(* Logix 5000 project; controller CarbonScout_MK6 vendor 1 type 14 code 154 rev 32.11; software revision 32.00; part 9 of 17 *)
(* tags used below, declared in another part *)
   AI_AIT_01 : P_AIn;   // pH
   AI_AIT_02 : P_AIn;   // DO
   AI_FIT_01 : P_AIn;   // Purge water flow
   AI_LIT_01 : P_AIn;   // Carbon Scout Laser Level Transmitter
   AI_LIT_02 : P_AIn;   // Carbon Scout Cone Level Transmitter
   AI_PIT_01 : P_AIn;   // Water supply pressure
   AI_WIT_01 : P_AIn;   // Weight measure
   CS_Alarms : P_Alarm[80];
   CS_DINTParams : DINT[100];
   CS_EventNum : DINT;
   CS_Result : CS_Results;   // Sample Result Live Async
   CS_Rules : DINT[17];
   CS_SampleSeq : DINT[129];
   CS_Seq : GEK_Sequence;
   CS_SeqCheckSum1 : DINT;
   CS_SeqCheckSum2 : DINT;
   CS_Tank : CS_TankParams[20];
   CS_TankOrder : DINT[17];
   CS_Timer : TIMER[80];
   CS_XRF : XRF;
   N50 : DINT[20];   // Out To Client (Ready only)
   N51 : DINT[5];   // From Client
   Oneshot : DINT;
   TankPointer : DINT;
   TimeAndDate : DINT[7];
   Valve_SPR_01 : P_ValveSO;   // Air injection valve
   Valve_XV_01 : P_ValveSO;   // Sample Valve Tank 1
   Valve_XV_02 : P_ValveSO;   // Sample Valve Tank 2
   Valve_XV_03 : P_ValveSO;   // Sample Valve Tank 3
   Valve_XV_04 : P_ValveSO;   // Sample Valve Tank 4
   Valve_XV_05 : P_ValveSO;   // Sample Valve Tank 5
   Valve_XV_06 : P_ValveSO;   // Sample Valve Tank 6
   Valve_XV_07 : P_ValveSO;   // Sample Valve Tank 7
   Valve_XV_08 : P_ValveSO;   // Sample Valve Tank 8
   Valve_XV_09 : P_ValveSO;   // Sample Valve Tank 9
   Valve_XV_10 : P_ValveSO;   // Sample Valve Tank 10
   Valve_XV_11 : P_ValveSO;   // Purge Valve
   Valve_XV_12 : P_ValveSO;   // Slurry inlet vavle
   Valve_XV_13 : P_ValveSO;   // Sample line vavle
   Valve_XV_14 : P_ValveSO;   // Top wash vavle
   Valve_XV_15 : P_ValveSO;   // Bottme wash vavle
   Valve_XV_16 : P_ValveSO;   // Potable water valve / Supply Water Valve
   Valve_XV_17 : P_ValveSO;   // Sample cone outlet vavle
   Valve_XV_18 : P_ValveSO;   // Sample strainer discharge
   Valve_XV_19 : P_ValveSO;   // Laser window
   Valve_XV_21_30 : P_ValveSO;   // Sample isolation valve
   Valve_XV_30 : P_ValveSO;   // XRF cooling valve
   Valve_XV_40 : P_ValveSO;   // XRF power on valve
(* DataMapping, continued *)

ROUTINE InputMapping   (* ladder *)
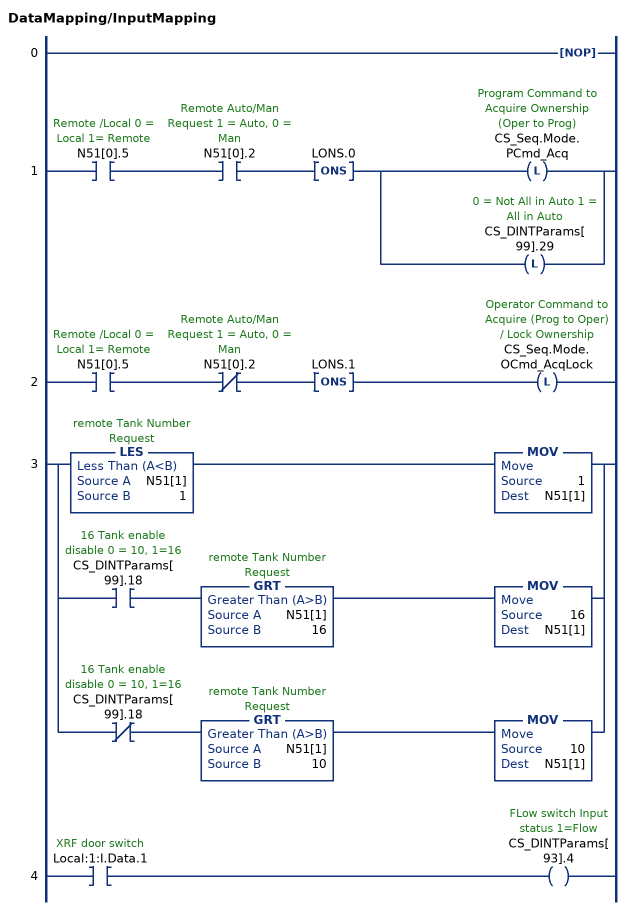
   0: NOP();
   1: XIC(N51[0].5)XIC(N51[0].2)ONS(LONS.0)[OTL(CS_Seq.Mode.PCmd_Acq) ,OTL(CS_DINTParams[99].29) ];
   2: XIC(N51[0].5)XIO(N51[0].2)ONS(LONS.1)OTL(CS_Seq.Mode.OCmd_AcqLock);
   3: [LES(N51[1],1) MOV(1,N51[1]) ,XIC(CS_DINTParams[99].18) GRT(N51[1],16) MOV(16,N51[1]) ,XIO(CS_DINTParams[99].18) GRT(N51[1],10) MOV(10,N51[1]) ];
   4: XIC(Local:1:I.Data.1)OTE(CS_DINTParams[93].4);
END_ROUTINE

ROUTINE Main   (* ladder *)
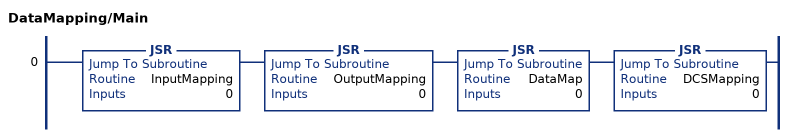
   0: JSR(InputMapping,0)JSR(OutputMapping,0)JSR(DataMap,0)JSR(DCSMapping,0);
END_ROUTINE

ROUTINE OutputMapping   (* ladder *)
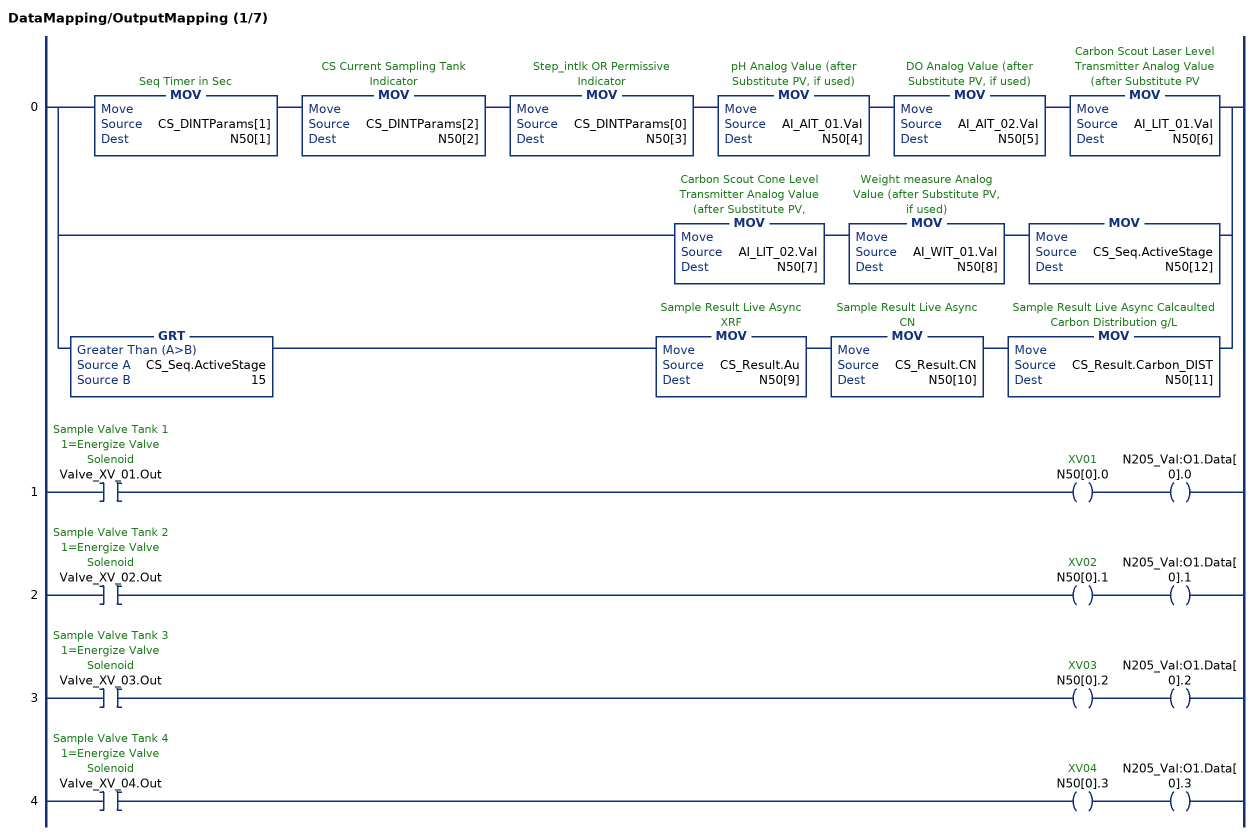
   0: [MOV(CS_DINTParams[1],N50[1]) MOV(CS_DINTParams[2],N50[2]) MOV(CS_DINTParams[0],N50[3]) MOV(AI_AIT_01.Val,N50[4]) MOV(AI_AIT_02.Val,N50[5]) MOV(AI_LIT_01.Val,N50[6]) ,MOV(AI_LIT_02.Val,N50[7]) MOV(AI_WIT_01.Val,N50[8]) MOV(CS_Seq.ActiveStage,N50[12]) ,GRT(CS_Seq.ActiveStage,15) MOV(CS_Result.Au,N50[9]) MOV(CS_Result.CN,N50[10]) MOV(CS_Result.Carbon_DIST,N50[11]) ];
   1: XIC(Valve_XV_01.Out)OTE(N50[0].0)OTE(N205_Val:O1.Data[0].0);
   2: XIC(Valve_XV_02.Out)OTE(N50[0].1)OTE(N205_Val:O1.Data[0].1);
   3: XIC(Valve_XV_03.Out)OTE(N50[0].2)OTE(N205_Val:O1.Data[0].2);
   4: XIC(Valve_XV_04.Out)OTE(N50[0].3)OTE(N205_Val:O1.Data[0].3);
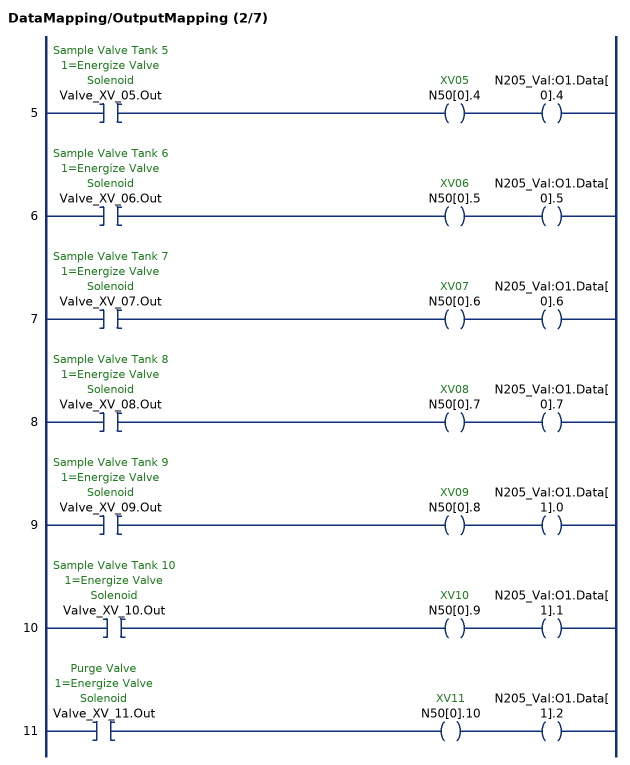
   5: XIC(Valve_XV_05.Out)OTE(N50[0].4)OTE(N205_Val:O1.Data[0].4);
   6: XIC(Valve_XV_06.Out)OTE(N50[0].5)OTE(N205_Val:O1.Data[0].5);
   7: XIC(Valve_XV_07.Out)OTE(N50[0].6)OTE(N205_Val:O1.Data[0].6);
   8: XIC(Valve_XV_08.Out)OTE(N50[0].7)OTE(N205_Val:O1.Data[0].7);
   9: XIC(Valve_XV_09.Out)OTE(N50[0].8)OTE(N205_Val:O1.Data[1].0);
   10: XIC(Valve_XV_10.Out)OTE(N50[0].9)OTE(N205_Val:O1.Data[1].1);
   11: XIC(Valve_XV_11.Out)OTE(N50[0].10)OTE(N205_Val:O1.Data[1].2);
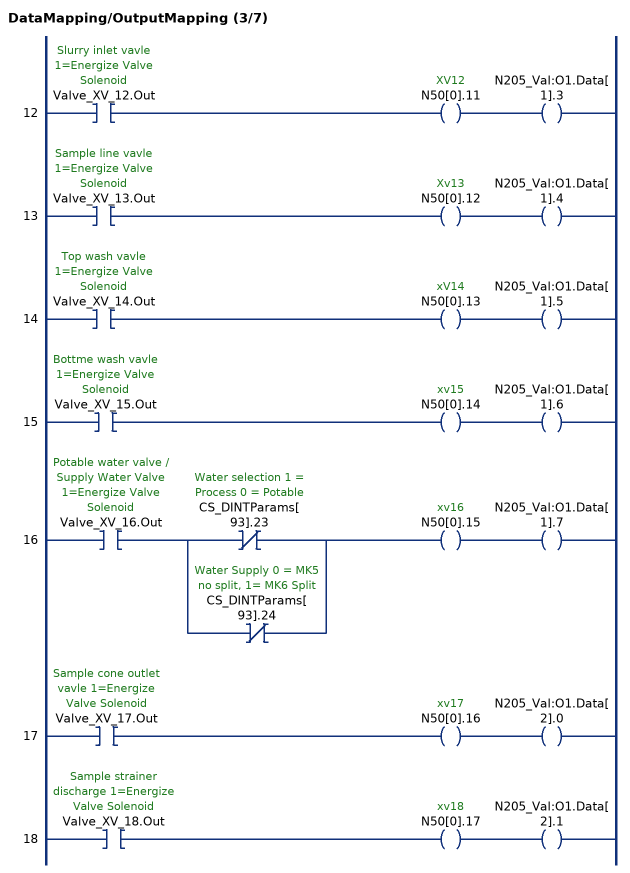
   12: XIC(Valve_XV_12.Out)OTE(N50[0].11)OTE(N205_Val:O1.Data[1].3);
   13: XIC(Valve_XV_13.Out)OTE(N50[0].12)OTE(N205_Val:O1.Data[1].4);
   14: XIC(Valve_XV_14.Out)OTE(N50[0].13)OTE(N205_Val:O1.Data[1].5);
   15: XIC(Valve_XV_15.Out)OTE(N50[0].14)OTE(N205_Val:O1.Data[1].6);
   16: XIC(Valve_XV_16.Out)[XIO(CS_DINTParams[93].23) ,XIO(CS_DINTParams[93].24) ]OTE(N50[0].15)OTE(N205_Val:O1.Data[1].7);
   17: XIC(Valve_XV_17.Out)OTE(N50[0].16)OTE(N205_Val:O1.Data[2].0);
   18: XIC(Valve_XV_18.Out)OTE(N50[0].17)OTE(N205_Val:O1.Data[2].1);
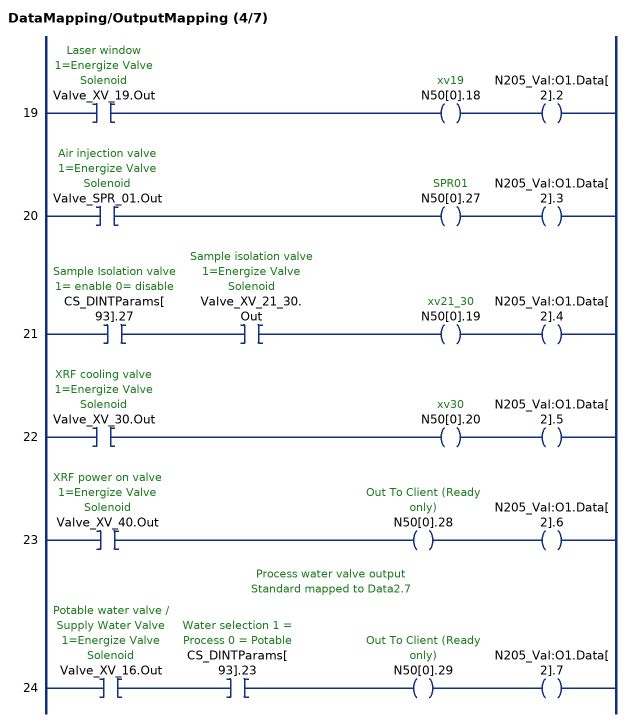
   19: XIC(Valve_XV_19.Out)OTE(N50[0].18)OTE(N205_Val:O1.Data[2].2);
   20: XIC(Valve_SPR_01.Out)OTE(N50[0].27)OTE(N205_Val:O1.Data[2].3);
   21: XIC(CS_DINTParams[93].27)XIC(Valve_XV_21_30.Out)OTE(N50[0].19)OTE(N205_Val:O1.Data[2].4);
   22: XIC(Valve_XV_30.Out)OTE(N50[0].20)OTE(N205_Val:O1.Data[2].5);
   23: XIC(Valve_XV_40.Out)OTE(N50[0].28)OTE(N205_Val:O1.Data[2].6);
   // Process water valve output
   // Standard mapped to Data2.7
   24: XIC(Valve_XV_16.Out)XIC(CS_DINTParams[93].23)OTE(N50[0].29)OTE(N205_Val:O1.Data[2].7);
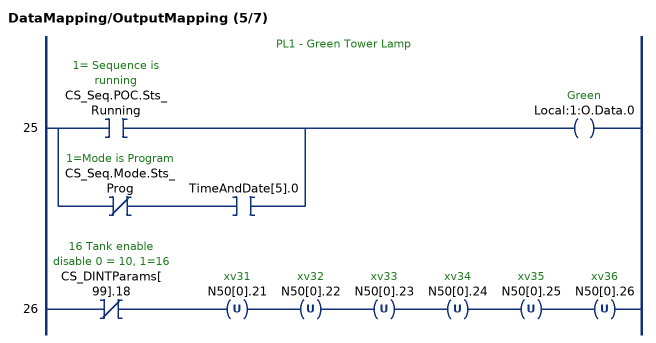
   // PL1 - Green Tower Lamp
   25: [XIC(CS_Seq.POC.Sts_Running) ,XIO(CS_Seq.Mode.Sts_Prog) XIC(TimeAndDate[5].0) ]OTE(Local:1:O.Data.0);
   26: XIO(CS_DINTParams[99].18)OTU(N50[0].21)OTU(N50[0].22)OTU(N50[0].23)OTU(N50[0].24)OTU(N50[0].25)OTU(N50[0].26);
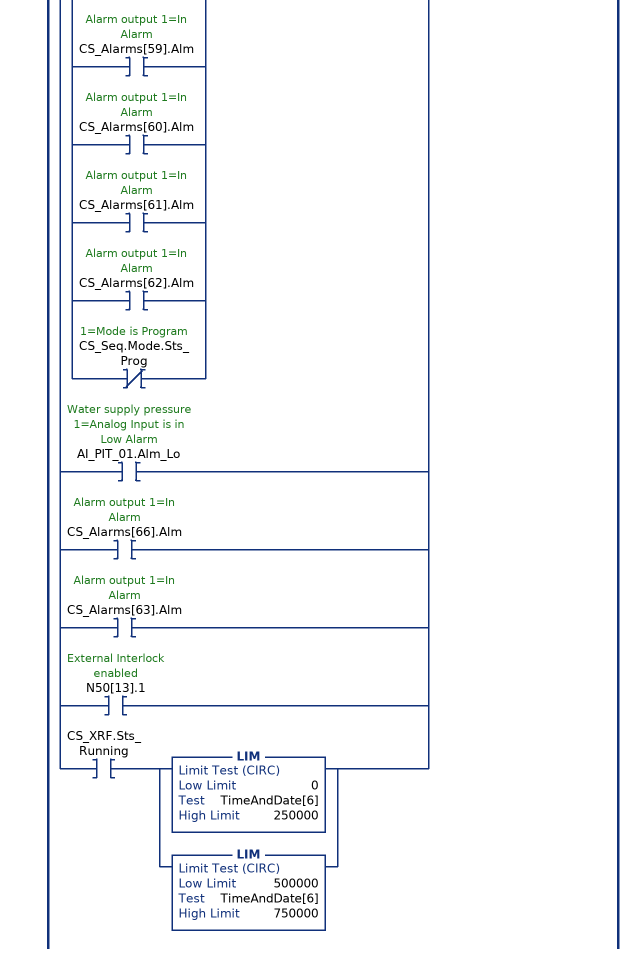
   // PL2 - Amber Tower Lamp
   27: [[XIC(CS_Alarms[24].Alm) ,XIC(CS_Alarms[14].Inp) ,XIC(CS_Alarms[15].Alm) ,XIC(CS_Alarms[16].Alm) ,XIC(CS_Alarms[17].Alm) ,XIC(CS_Alarms[18].Alm) ,XIC(CS_Alarms[19].Alm) ,XIC(CS_Alarms[20].Alm) ,XIC(CS_Alarms[21].Alm) ,XIC(CS_Alarms[22].Alm) ,XIC(CS_Alarms[23].Alm) ,XIC(CS_Alarms[57].Alm) ,XIC(CS_Alarms[58].Alm) ,XIC(CS_Alarms[59].Alm) ,XIC(CS_Alarms[60].Alm) ,XIC(CS_Alarms[61].Alm) ,XIC(CS_Alarms[62].Alm) ,XIO(CS_Seq.Mode.Sts_Prog) ] XIC(TimeAndDate[5].0) XIO(CS_XRF.Sts_Running) ,XIC(AI_PIT_01.Alm_Lo) ,XIC(CS_Alarms[66].Alm) ,XIC(CS_Alarms[63].Alm) ,XIC(N50[13].1) ,XIC(CS_XRF.Sts_Running) [LIM(0,TimeAndDate[6],250000) ,LIM(500000,TimeAndDate[6],750000) ] ]OTE(Local:1:O.Data.1);
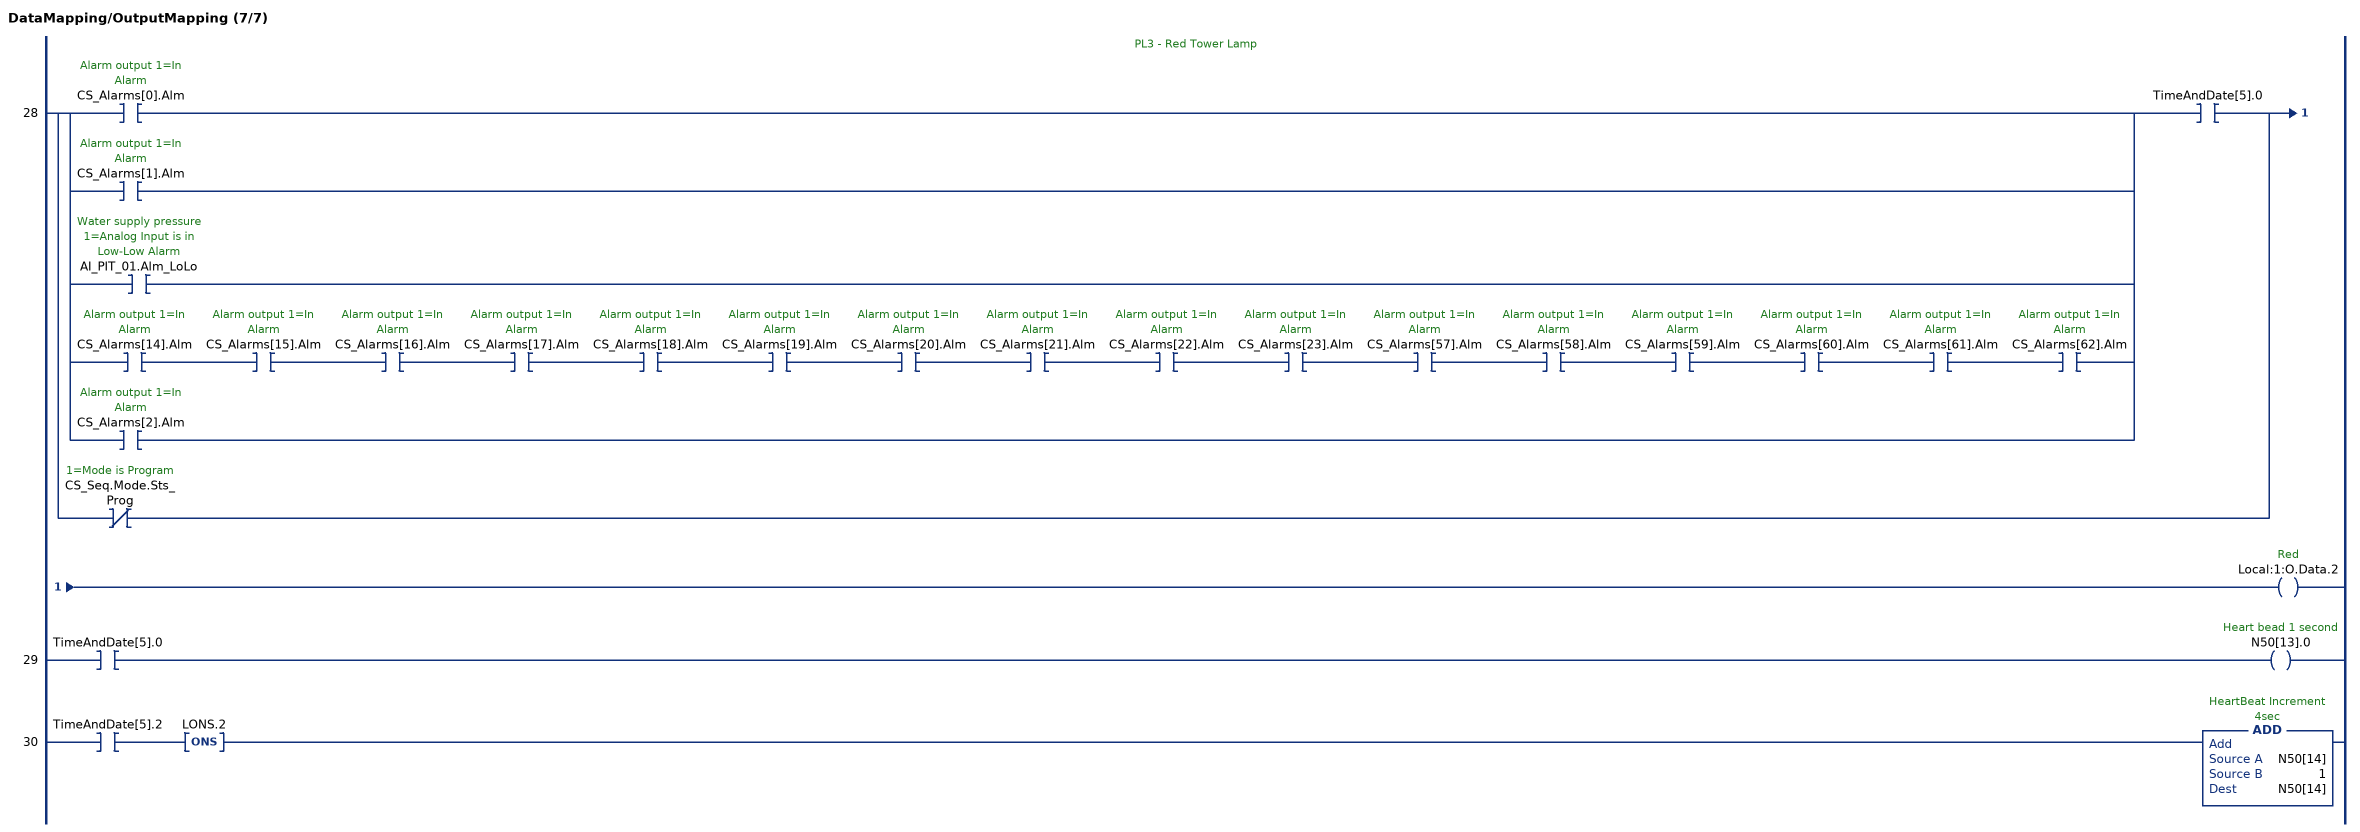
   // PL3 - Red Tower Lamp
   28: [[XIC(CS_Alarms[0].Alm) ,XIC(CS_Alarms[1].Alm) ,XIC(AI_PIT_01.Alm_LoLo) ,XIC(CS_Alarms[14].Alm) XIC(CS_Alarms[15].Alm) XIC(CS_Alarms[16].Alm) XIC(CS_Alarms[17].Alm) XIC(CS_Alarms[18].Alm) XIC(CS_Alarms[19].Alm) XIC(CS_Alarms[20].Alm) XIC(CS_Alarms[21].Alm) XIC(CS_Alarms[22].Alm) XIC(CS_Alarms[23].Alm) XIC(CS_Alarms[57].Alm) XIC(CS_Alarms[58].Alm) XIC(CS_Alarms[59].Alm) XIC(CS_Alarms[60].Alm) XIC(CS_Alarms[61].Alm) XIC(CS_Alarms[62].Alm) ,XIC(CS_Alarms[2].Alm) ] XIC(TimeAndDate[5].0) ,XIO(CS_Seq.Mode.Sts_Prog) ]OTE(Local:1:O.Data.2);
   29: XIC(TimeAndDate[5].0)OTE(N50[13].0);
   30: XIC(TimeAndDate[5].2)ONS(LONS.2)ADD(N50[14],1,N50[14]);
END_ROUTINE
END_PROGRAM

PROGRAM Powerup   (* main routine Yes *)
VAR
   ControllerFaultReset : DINT;
   MajorFaultBit : DINT;
   MajorFaultEvent : DINT;
   MinorEvents : DINT;
   MinorFaultBits : DINT;
END_VAR

ROUTINE Yes   (* ladder *)
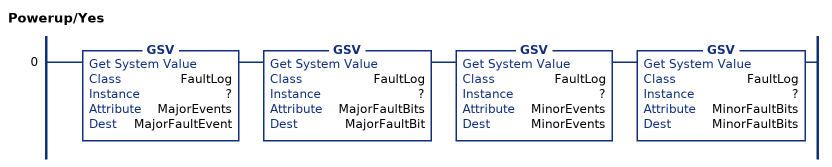
   0: GSV(FaultLog,?,MajorEvents,MajorFaultEvent)GSV(FaultLog,?,MajorFaultBits,MajorFaultBit)GSV(FaultLog,?,MinorEvents,MinorEvents)GSV(FaultLog,?,MinorFaultBits,MinorFaultBits);
END_ROUTINE
END_PROGRAM

PROGRAM SeqProgram   (* main routine MainRoutine *)
VAR
   CNT : DINT := 311;
   CS_EVentNumStore : DINT := 1;
   Data_TLSaver : BOOL := 1;
   Delay : TIMER := (PRE := 10000);
   DN_Cal : BOOL;   // Calculation Done Bit to proceed next step
   EventDone : BOOL;
   ExtraValveCNTReached : BOOL; {access Read Only}
   ExtraValvesAuto : BOOL; {access Read Only}
   i : DINT;
   Index : DINT := 1;
   IndexNumStore : DINT := 8;
   InitialPurgeRequired : BOOL := 1;
   LIT_Prev : REAL := 1441.9149;
   LocalSampleTank : DINT := 6;
   LOnlineNumber : DINT := 7;
   LONS : DINT := 1;
   ManualRunning : BOOL;
   MaxFindIndexNum : DINT := 16;
   MaxFindNum : DINT := 1;
   ONS : BOOL[32] := ([1] := 1, [4] := 1);
   SampleIndexNum : DINT := 8;
   SampleIndexNum2 : DINT;
   SONS : DINT := 511;
   storage : BOOL;
   TankDiagnosticCheck : BOOL;
   TimeCompare : TimerCompare := (In_PresetTime1_Multiplier := 60, In_PresetTime2 := 10, In_PresetTime2_Multiplier := 1, In_ActiveStep := 23);
   TimeRemainingCal : TimeRemainingCal := (In_PresetTime := 30, RemainingSec := 8, In_Time := 1);
   XRF_DirtyWinCounter : COUNTER := (PRE := 10);
   XRF_ReadyTimer : TIMER := (PRE := 10000);
END_VAR

ROUTINE _SampleSeq   (* ladder *)
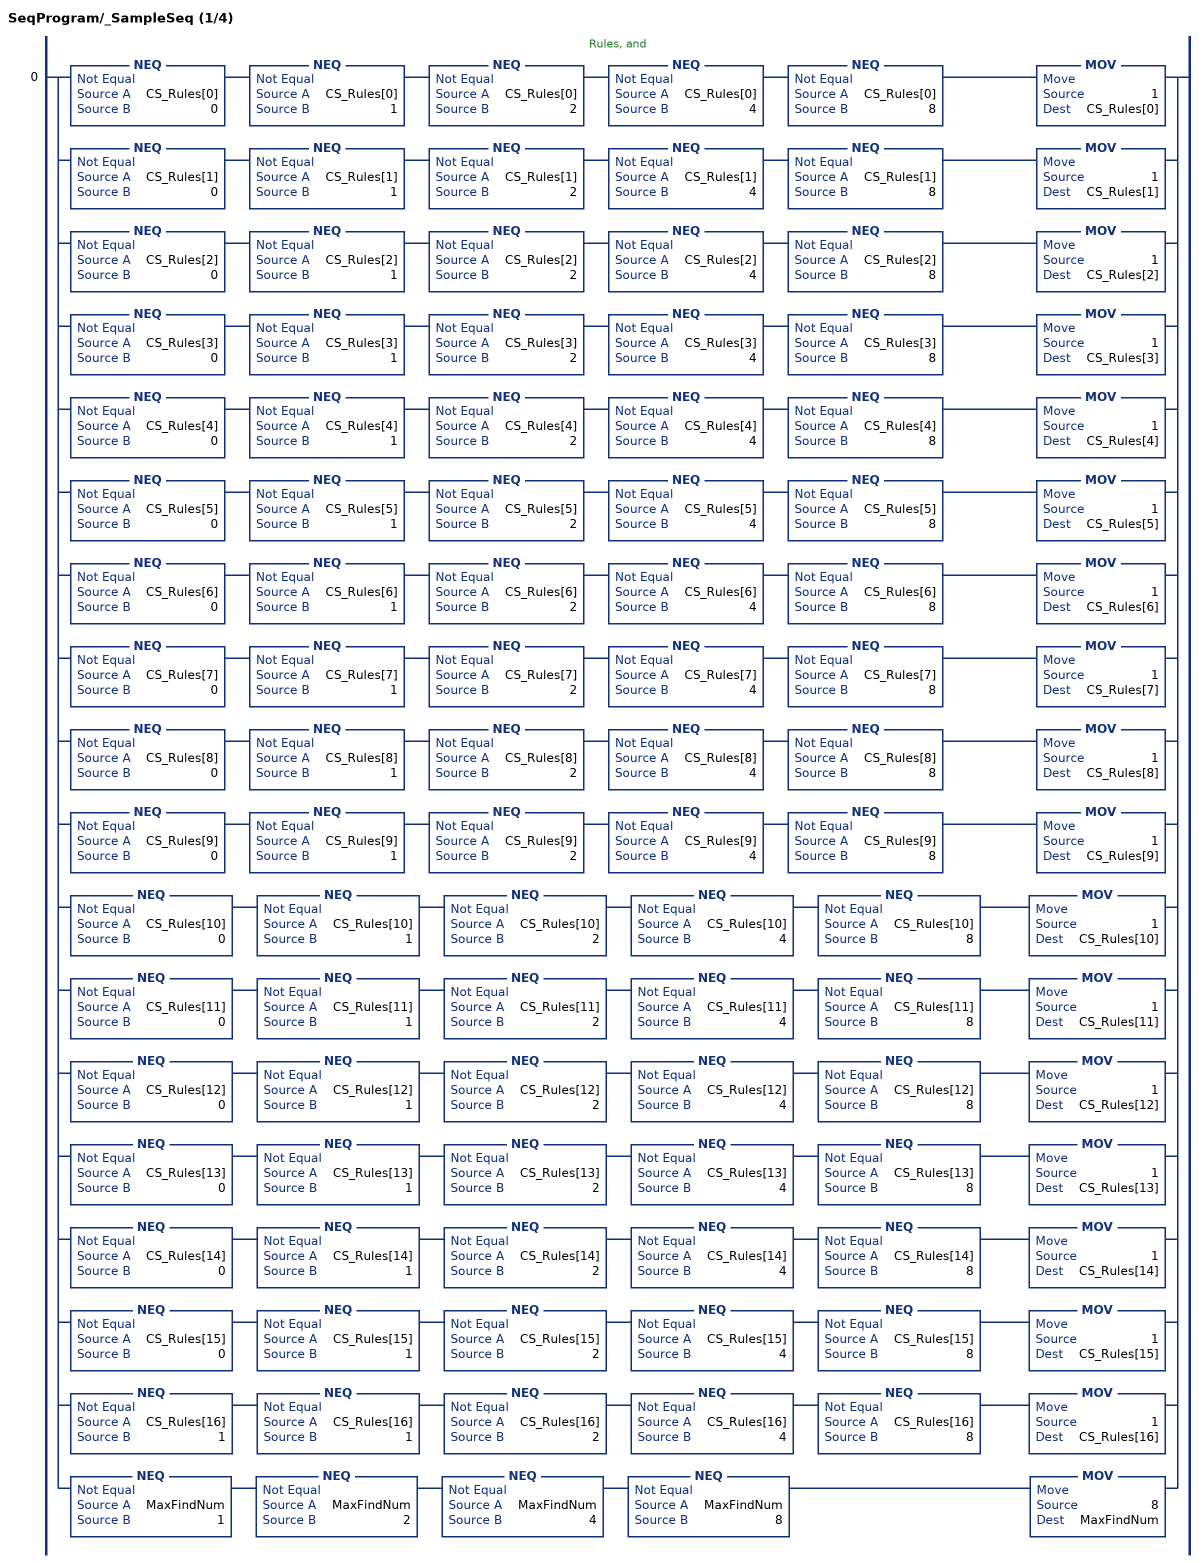
   // Rules, and
   0: [NEQ(CS_Rules[0],0) NEQ(CS_Rules[0],1) NEQ(CS_Rules[0],2) NEQ(CS_Rules[0],4) NEQ(CS_Rules[0],8) MOV(1,CS_Rules[0]) ,NEQ(CS_Rules[1],0) NEQ(CS_Rules[1],1) NEQ(CS_Rules[1],2) NEQ(CS_Rules[1],4) NEQ(CS_Rules[1],8) MOV(1,CS_Rules[1]) ,NEQ(CS_Rules[2],0) NEQ(CS_Rules[2],1) NEQ(CS_Rules[2],2) NEQ(CS_Rules[2],4) NEQ(CS_Rules[2],8) MOV(1,CS_Rules[2]) ,NEQ(CS_Rules[3],0) NEQ(CS_Rules[3],1) NEQ(CS_Rules[3],2) NEQ(CS_Rules[3],4) NEQ(CS_Rules[3],8) MOV(1,CS_Rules[3]) ,NEQ(CS_Rules[4],0) NEQ(CS_Rules[4],1) NEQ(CS_Rules[4],2) NEQ(CS_Rules[4],4) NEQ(CS_Rules[4],8) MOV(1,CS_Rules[4]) ,NEQ(CS_Rules[5],0) NEQ(CS_Rules[5],1) NEQ(CS_Rules[5],2) NEQ(CS_Rules[5],4) NEQ(CS_Rules[5],8) MOV(1,CS_Rules[5]) ,NEQ(CS_Rules[6],0) NEQ(CS_Rules[6],1) NEQ(CS_Rules[6],2) NEQ(CS_Rules[6],4) NEQ(CS_Rules[6],8) MOV(1,CS_Rules[6]) ,NEQ(CS_Rules[7],0) NEQ(CS_Rules[7],1) NEQ(CS_Rules[7],2) NEQ(CS_Rules[7],4) NEQ(CS_Rules[7],8) MOV(1,CS_Rules[7]) ,NEQ(CS_Rules[8],0) NEQ(CS_Rules[8],1) NEQ(CS_Rules[8],2) NEQ(CS_Rules[8],4) NEQ(CS_Rules[8],8) MOV(1,CS_Rules[8]) ,NEQ(CS_Rules[9],0) NEQ(CS_Rules[9],1) NEQ(CS_Rules[9],2) NEQ(CS_Rules[9],4) NEQ(CS_Rules[9],8) MOV(1,CS_Rules[9]) ,NEQ(CS_Rules[10],0) NEQ(CS_Rules[10],1) NEQ(CS_Rules[10],2) NEQ(CS_Rules[10],4) NEQ(CS_Rules[10],8) MOV(1,CS_Rules[10]) ,NEQ(CS_Rules[11],0) NEQ(CS_Rules[11],1) NEQ(CS_Rules[11],2) NEQ(CS_Rules[11],4) NEQ(CS_Rules[11],8) MOV(1,CS_Rules[11]) ,NEQ(CS_Rules[12],0) NEQ(CS_Rules[12],1) NEQ(CS_Rules[12],2) NEQ(CS_Rules[12],4) NEQ(CS_Rules[12],8) MOV(1,CS_Rules[12]) ,NEQ(CS_Rules[13],0) NEQ(CS_Rules[13],1) NEQ(CS_Rules[13],2) NEQ(CS_Rules[13],4) NEQ(CS_Rules[13],8) MOV(1,CS_Rules[13]) ,NEQ(CS_Rules[14],0) NEQ(CS_Rules[14],1) NEQ(CS_Rules[14],2) NEQ(CS_Rules[14],4) NEQ(CS_Rules[14],8) MOV(1,CS_Rules[14]) ,NEQ(CS_Rules[15],0) NEQ(CS_Rules[15],1) NEQ(CS_Rules[15],2) NEQ(CS_Rules[15],4) NEQ(CS_Rules[15],8) MOV(1,CS_Rules[15]) ,NEQ(CS_Rules[16],1) NEQ(CS_Rules[16],1) NEQ(CS_Rules[16],2) NEQ(CS_Rules[16],4) NEQ(CS_Rules[16],8) MOV(1,CS_Rules[16]) ,NEQ(MaxFindNum,1) NEQ(MaxFindNum,2) NEQ(MaxFindNum,4) NEQ(MaxFindNum,8) MOV(8,MaxFindNum) ];
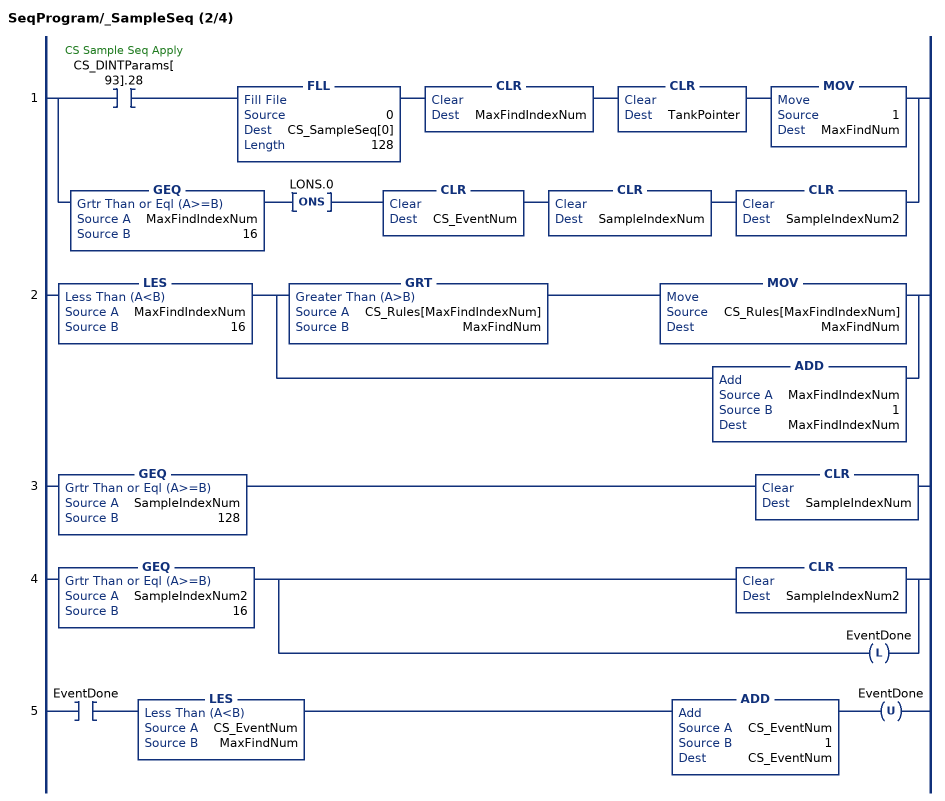
   1: [XIC(CS_DINTParams[93].28) FLL(0,CS_SampleSeq[0],128) CLR(MaxFindIndexNum) CLR(TankPointer) MOV(1,MaxFindNum) ,GEQ(MaxFindIndexNum,16) ONS(LONS.0) CLR(CS_EventNum) CLR(SampleIndexNum) CLR(SampleIndexNum2) ];
   2: LES(MaxFindIndexNum,16)[GRT(CS_Rules[MaxFindIndexNum],MaxFindNum) MOV(CS_Rules[MaxFindIndexNum],MaxFindNum) ,ADD(MaxFindIndexNum,1,MaxFindIndexNum) ];
   3: GEQ(SampleIndexNum,128)CLR(SampleIndexNum);
   4: GEQ(SampleIndexNum2,16)[CLR(SampleIndexNum2) ,OTL(EventDone) ];
   5: XIC(EventDone)LES(CS_EventNum,MaxFindNum)ADD(CS_EventNum,1,CS_EventNum)OTU(EventDone);
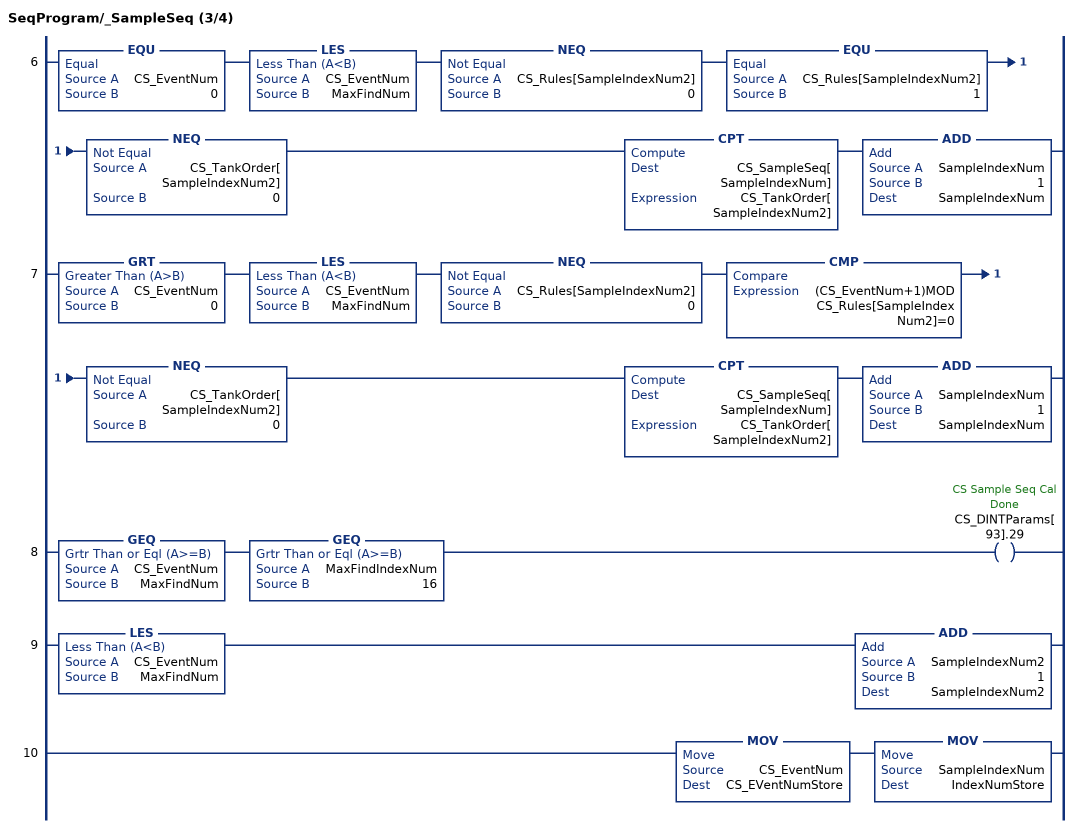
   6: EQU(CS_EventNum,0)LES(CS_EventNum,MaxFindNum)NEQ(CS_Rules[SampleIndexNum2],0)EQU(CS_Rules[SampleIndexNum2],1)NEQ(CS_TankOrder[SampleIndexNum2],0)CPT(CS_SampleSeq[SampleIndexNum],CS_TankOrder[SampleIndexNum2])ADD(SampleIndexNum,1,SampleIndexNum);
   7: GRT(CS_EventNum,0)LES(CS_EventNum,MaxFindNum)NEQ(CS_Rules[SampleIndexNum2],0)CMP((CS_EventNum+1)MOD CS_Rules[SampleIndexNum2]=0)NEQ(CS_TankOrder[SampleIndexNum2],0)CPT(CS_SampleSeq[SampleIndexNum],CS_TankOrder[SampleIndexNum2])ADD(SampleIndexNum,1,SampleIndexNum);
   8: GEQ(CS_EventNum,MaxFindNum)GEQ(MaxFindIndexNum,16)OTE(CS_DINTParams[93].29);
   9: LES(CS_EventNum,MaxFindNum)ADD(SampleIndexNum2,1,SampleIndexNum2);
   10: MOV(CS_EventNum,CS_EVentNumStore)MOV(SampleIndexNum,IndexNumStore);
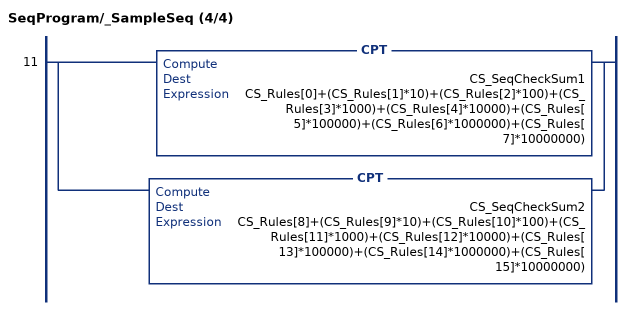
   11: [CPT(CS_SeqCheckSum1,CS_Rules[0]+(CS_Rules[1]*10)+(CS_Rules[2]*100)+(CS_Rules[3]*1000)+(CS_Rules[4]*10000)+(CS_Rules[5]*100000)+(CS_Rules[6]*1000000)+(CS_Rules[7]*10000000)) ,CPT(CS_SeqCheckSum2,CS_Rules[8]+(CS_Rules[9]*10)+(CS_Rules[10]*100)+(CS_Rules[11]*1000)+(CS_Rules[12]*10000)+(CS_Rules[13]*100000)+(CS_Rules[14]*1000000)+(CS_Rules[15]*10000000)) ];
END_ROUTINE

ROUTINE Alarms   (* ladder *)
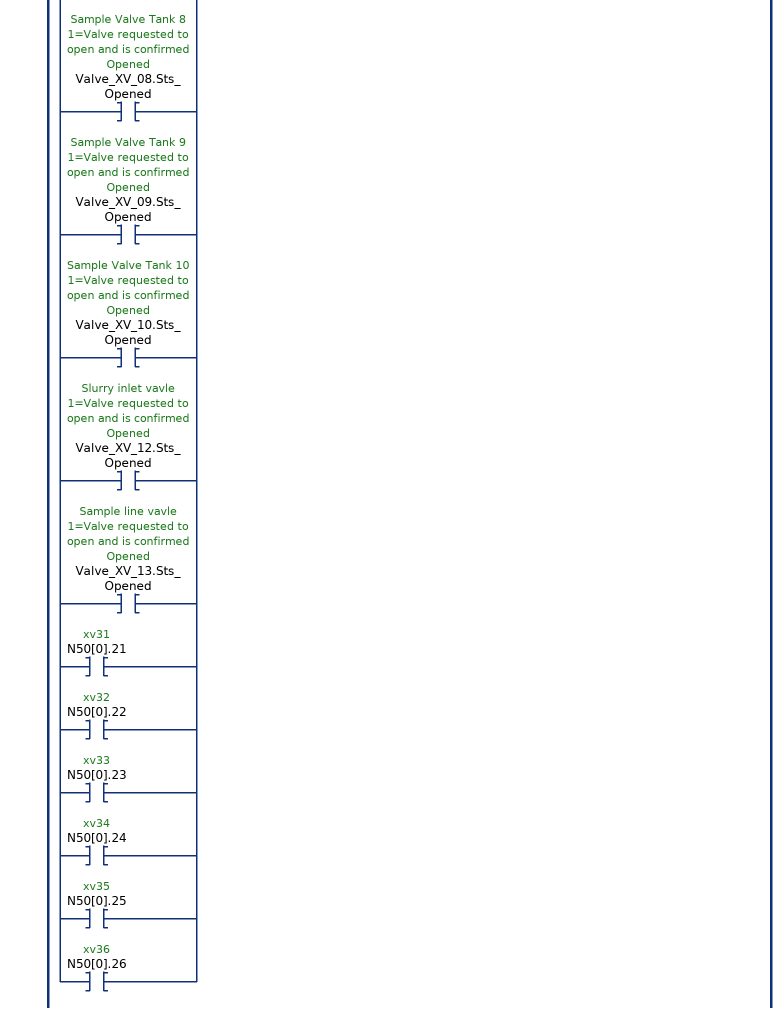
   0: [XIC(Valve_XV_01.Sts_Opened) ,XIC(Valve_XV_12.Sts_Opened) ,XIC(Valve_XV_02.Sts_Opened) ,XIC(Valve_XV_03.Sts_Opened) ,XIC(Valve_XV_04.Sts_Opened) ,XIC(Valve_XV_05.Sts_Opened) ,XIC(Valve_XV_06.Sts_Opened) ,XIC(Valve_XV_07.Sts_Opened) ,XIC(Valve_XV_08.Sts_Opened) ,XIC(Valve_XV_09.Sts_Opened) ,XIC(Valve_XV_10.Sts_Opened) ,XIC(Valve_XV_12.Sts_Opened) ,XIC(Valve_XV_13.Sts_Opened) ,XIC(N50[0].21) ,XIC(N50[0].22) ,XIC(N50[0].23) ,XIC(N50[0].24) ,XIC(N50[0].25) ,XIC(N50[0].26) ]XIC(Valve_XV_11.Sts_Opened)XIO(CS_DINTParams[93].0)OTE(AI_FIT_01.Inp_LoGate)OTE(AI_FIT_01.Inp_LoLoGate);
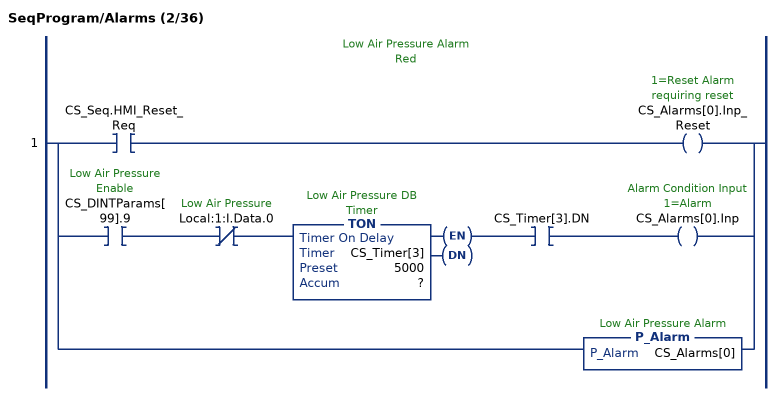
   // Low Air Pressure Alarm
   // Red
   1: [XIC(CS_Seq.HMI_Reset_Req) OTE(CS_Alarms[0].Inp_Reset) ,XIC(CS_DINTParams[99].9) XIO(Local:1:I.Data.0) TON(CS_Timer[3],?,?) XIC(CS_Timer[3].DN) OTE(CS_Alarms[0].Inp) ,P_Alarm(CS_Alarms[0]) ];
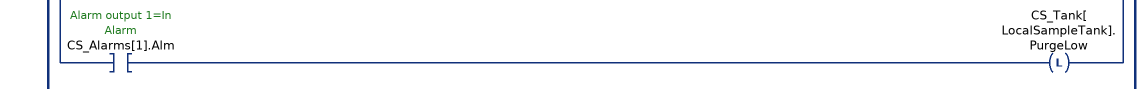
   // Purge Water Flow Alarm
   // Amber
   2: [XIC(CS_Seq.HMI_Reset_Req) OTE(CS_Alarms[1].Inp_Reset) ,[XIC(Valve_XV_01.Sts_Opened) ,XIC(Valve_XV_02.Sts_Opened) ,XIC(Valve_XV_03.Sts_Opened) ,XIC(Valve_XV_04.Sts_Opened) ,XIC(Valve_XV_05.Sts_Opened) ,XIC(Valve_XV_06.Sts_Opened) ,XIC(Valve_XV_07.Sts_Opened) ,XIC(Valve_XV_08.Sts_Opened) ,XIC(Valve_XV_09.Sts_Opened) ,XIC(Valve_XV_10.Sts_Opened) ,XIC(Valve_XV_12.Sts_Opened) ,XIC(Valve_XV_13.Sts_Opened) ,XIC(N50[0].21) ,XIC(N50[0].22) ,XIC(N50[0].23) ,XIC(N50[0].24) ,XIC(N50[0].25) ,XIC(N50[0].26) ] XIC(Valve_XV_11.Sts_Opened) [XIC(AI_FIT_01.Alm_Lo) XIO(CS_DINTParams[93].0) ,XIC(AI_FIT_01.Alm_LoLo) XIO(CS_DINTParams[93].0) ,XIO(Local:1:I.Data.1) XIC(CS_DINTParams[93].0) ] TON(CS_Timer[4],?,?) XIC(CS_Timer[4].DN) OTE(CS_Alarms[1].Inp) ,P_Alarm(CS_Alarms[1]) ,XIC(CS_Alarms[1].Alm) OTL(CS_Tank[LocalSampleTank].PurgeLow) ];
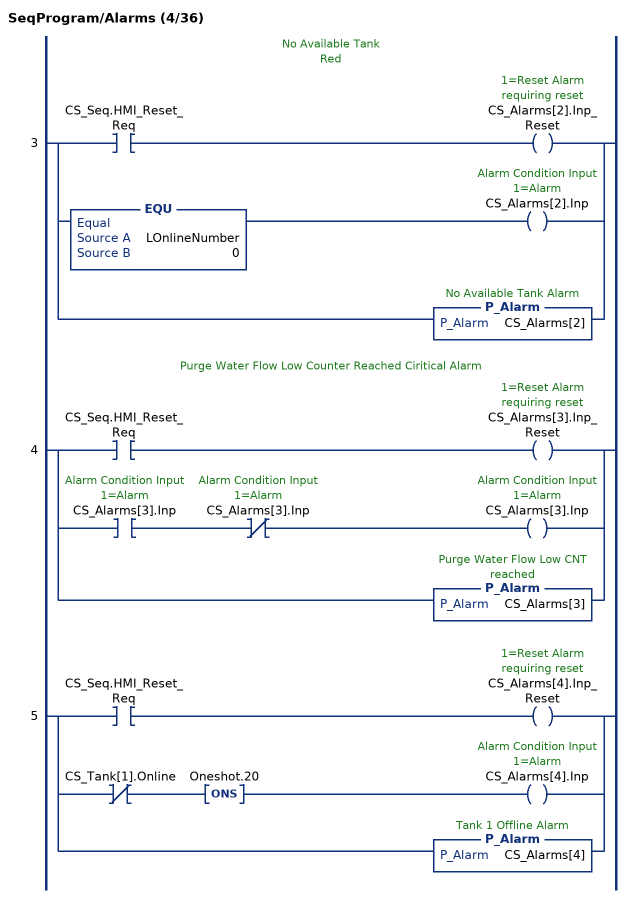
   // No Available Tank
   // Red
   3: [XIC(CS_Seq.HMI_Reset_Req) OTE(CS_Alarms[2].Inp_Reset) ,EQU(LOnlineNumber,0) OTE(CS_Alarms[2].Inp) ,P_Alarm(CS_Alarms[2]) ];
   // Purge Water Flow Low Counter Reached Ciritical Alarm
   4: [XIC(CS_Seq.HMI_Reset_Req) OTE(CS_Alarms[3].Inp_Reset) ,XIC(CS_Alarms[3].Inp) XIO(CS_Alarms[3].Inp) OTE(CS_Alarms[3].Inp) ,P_Alarm(CS_Alarms[3]) ];
   5: [XIC(CS_Seq.HMI_Reset_Req) OTE(CS_Alarms[4].Inp_Reset) ,XIO(CS_Tank[1].Online) ONS(Oneshot.20) OTE(CS_Alarms[4].Inp) ,P_Alarm(CS_Alarms[4]) ];
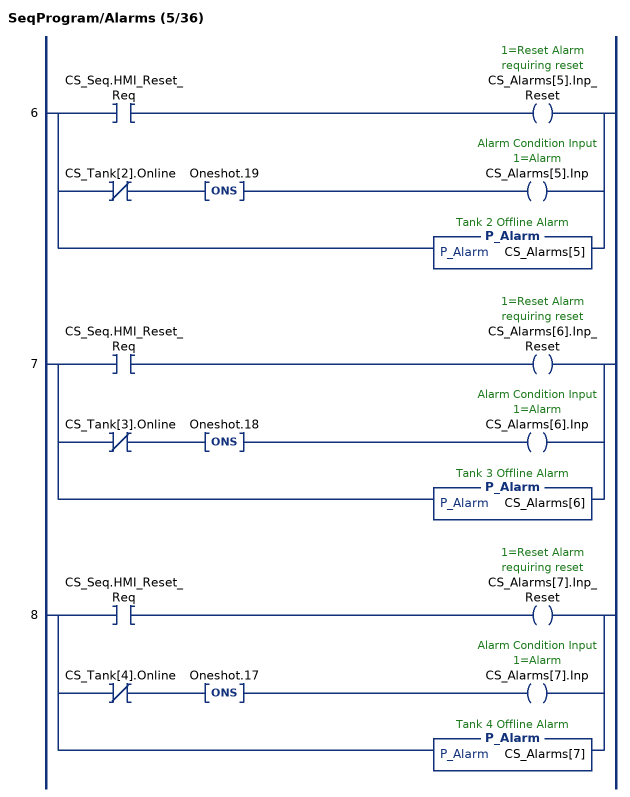
   6: [XIC(CS_Seq.HMI_Reset_Req) OTE(CS_Alarms[5].Inp_Reset) ,XIO(CS_Tank[2].Online) ONS(Oneshot.19) OTE(CS_Alarms[5].Inp) ,P_Alarm(CS_Alarms[5]) ];
   7: [XIC(CS_Seq.HMI_Reset_Req) OTE(CS_Alarms[6].Inp_Reset) ,XIO(CS_Tank[3].Online) ONS(Oneshot.18) OTE(CS_Alarms[6].Inp) ,P_Alarm(CS_Alarms[6]) ];
   8: [XIC(CS_Seq.HMI_Reset_Req) OTE(CS_Alarms[7].Inp_Reset) ,XIO(CS_Tank[4].Online) ONS(Oneshot.17) OTE(CS_Alarms[7].Inp) ,P_Alarm(CS_Alarms[7]) ];
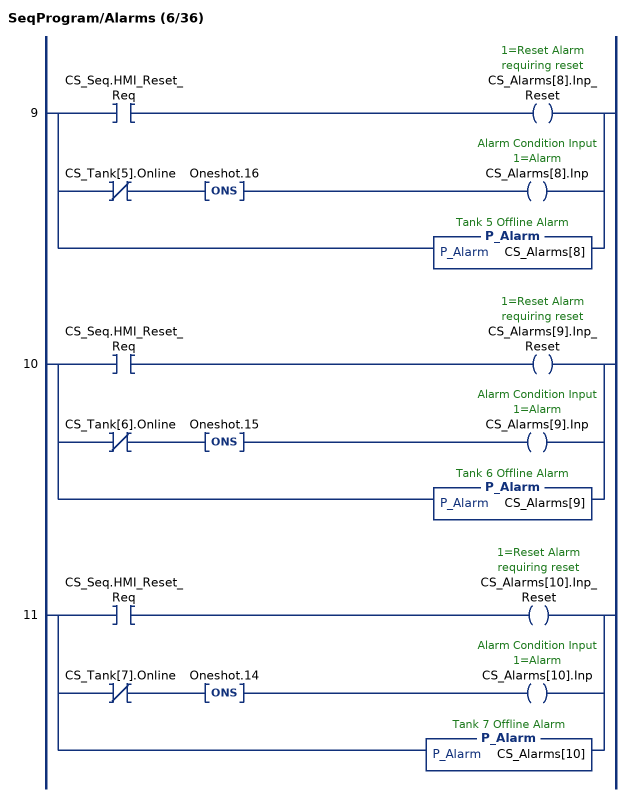
   9: [XIC(CS_Seq.HMI_Reset_Req) OTE(CS_Alarms[8].Inp_Reset) ,XIO(CS_Tank[5].Online) ONS(Oneshot.16) OTE(CS_Alarms[8].Inp) ,P_Alarm(CS_Alarms[8]) ];
   10: [XIC(CS_Seq.HMI_Reset_Req) OTE(CS_Alarms[9].Inp_Reset) ,XIO(CS_Tank[6].Online) ONS(Oneshot.15) OTE(CS_Alarms[9].Inp) ,P_Alarm(CS_Alarms[9]) ];
   11: [XIC(CS_Seq.HMI_Reset_Req) OTE(CS_Alarms[10].Inp_Reset) ,XIO(CS_Tank[7].Online) ONS(Oneshot.14) OTE(CS_Alarms[10].Inp) ,P_Alarm(CS_Alarms[10]) ];
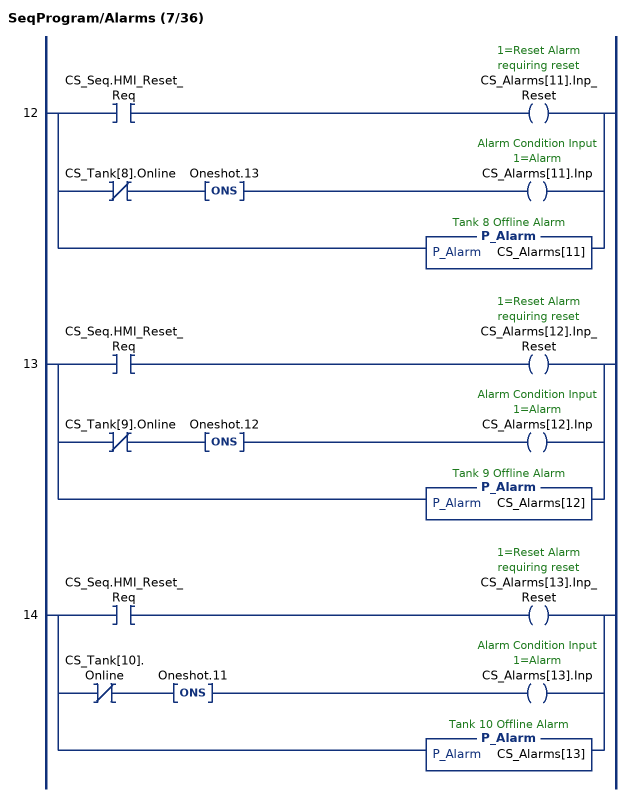
   12: [XIC(CS_Seq.HMI_Reset_Req) OTE(CS_Alarms[11].Inp_Reset) ,XIO(CS_Tank[8].Online) ONS(Oneshot.13) OTE(CS_Alarms[11].Inp) ,P_Alarm(CS_Alarms[11]) ];
   13: [XIC(CS_Seq.HMI_Reset_Req) OTE(CS_Alarms[12].Inp_Reset) ,XIO(CS_Tank[9].Online) ONS(Oneshot.12) OTE(CS_Alarms[12].Inp) ,P_Alarm(CS_Alarms[12]) ];
   14: [XIC(CS_Seq.HMI_Reset_Req) OTE(CS_Alarms[13].Inp_Reset) ,XIO(CS_Tank[10].Online) ONS(Oneshot.11) OTE(CS_Alarms[13].Inp) ,P_Alarm(CS_Alarms[13]) ];
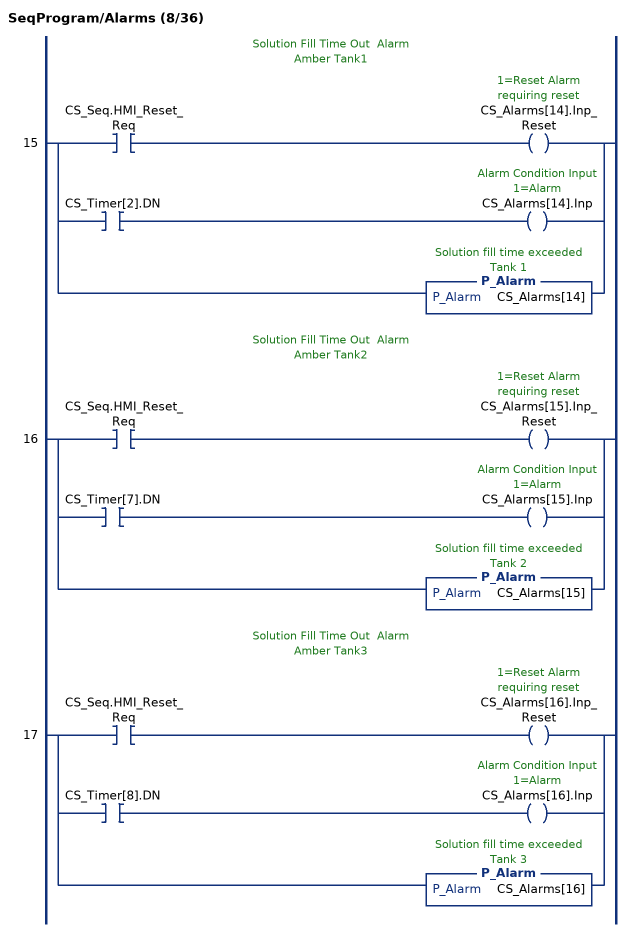
   // Solution Fill Time Out  Alarm
   // Amber Tank1
   15: [XIC(CS_Seq.HMI_Reset_Req) OTE(CS_Alarms[14].Inp_Reset) ,XIC(CS_Timer[2].DN) OTE(CS_Alarms[14].Inp) ,P_Alarm(CS_Alarms[14]) ];
   // Solution Fill Time Out  Alarm
   // Amber Tank2
   16: [XIC(CS_Seq.HMI_Reset_Req) OTE(CS_Alarms[15].Inp_Reset) ,XIC(CS_Timer[7].DN) OTE(CS_Alarms[15].Inp) ,P_Alarm(CS_Alarms[15]) ];
   // Solution Fill Time Out  Alarm
   // Amber Tank3
   17: [XIC(CS_Seq.HMI_Reset_Req) OTE(CS_Alarms[16].Inp_Reset) ,XIC(CS_Timer[8].DN) OTE(CS_Alarms[16].Inp) ,P_Alarm(CS_Alarms[16]) ];
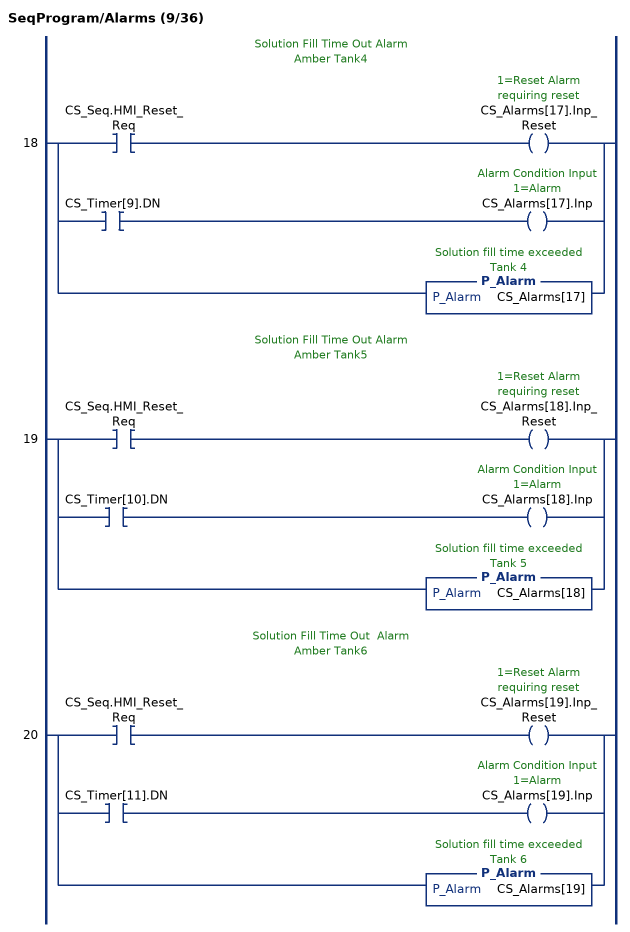
   // Solution Fill Time Out Alarm
   // Amber Tank4
   18: [XIC(CS_Seq.HMI_Reset_Req) OTE(CS_Alarms[17].Inp_Reset) ,XIC(CS_Timer[9].DN) OTE(CS_Alarms[17].Inp) ,P_Alarm(CS_Alarms[17]) ];
   // Solution Fill Time Out Alarm
   // Amber Tank5
   19: [XIC(CS_Seq.HMI_Reset_Req) OTE(CS_Alarms[18].Inp_Reset) ,XIC(CS_Timer[10].DN) OTE(CS_Alarms[18].Inp) ,P_Alarm(CS_Alarms[18]) ];
   // Solution Fill Time Out  Alarm
   // Amber Tank6
   20: [XIC(CS_Seq.HMI_Reset_Req) OTE(CS_Alarms[19].Inp_Reset) ,XIC(CS_Timer[11].DN) OTE(CS_Alarms[19].Inp) ,P_Alarm(CS_Alarms[19]) ];
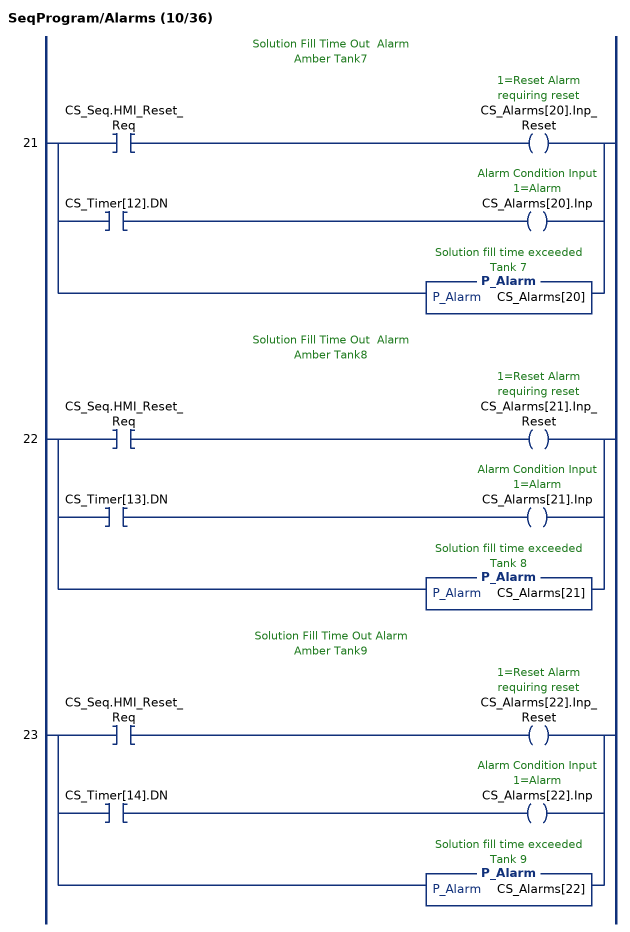
   // Solution Fill Time Out  Alarm
   // Amber Tank7
   21: [XIC(CS_Seq.HMI_Reset_Req) OTE(CS_Alarms[20].Inp_Reset) ,XIC(CS_Timer[12].DN) OTE(CS_Alarms[20].Inp) ,P_Alarm(CS_Alarms[20]) ];
   // Solution Fill Time Out  Alarm
   // Amber Tank8
   22: [XIC(CS_Seq.HMI_Reset_Req) OTE(CS_Alarms[21].Inp_Reset) ,XIC(CS_Timer[13].DN) OTE(CS_Alarms[21].Inp) ,P_Alarm(CS_Alarms[21]) ];
   // Solution Fill Time Out Alarm
   // Amber Tank9
   23: [XIC(CS_Seq.HMI_Reset_Req) OTE(CS_Alarms[22].Inp_Reset) ,XIC(CS_Timer[14].DN) OTE(CS_Alarms[22].Inp) ,P_Alarm(CS_Alarms[22]) ];
